Yaskawa INFORM job: X2_48(150,-90).JBI

/JOB
//NAME X2_48(150,-90)
//POS
///NPOS 103,103,103,5,0,0
///TOOL 0
///POSTYPE PULSE
///PULSE
C00000=-2000,-112988,-119327,0,83158,0
C00001=142756,-112988,-119327,18089,83158,-34222
C00002=145489,-137180,-128771,21394,87700,-32111
C00003=164591,-94889,-79086,18920,74682,-27376
C00004=167906,-89992,-74155,18360,73432,-26351
C00005=169175,-88015,-72150,18139,72941,-25959
C00006=169090,-86796,-69106,18271,71772,-26171
C00007=169175,-88015,-72150,18139,72941,-25959
C00008=170099,-88727,-72164,17993,72396,-25701
C00009=172764,-85592,-70856,17391,72586,-24688
C00010=170099,-88727,-72164,17993,72396,-25701
C00011=185420,-95958,-68594,-7326,50076,-11474
C00012=182716,-92695,-67464,-5857,50831,-12695
C00013=185420,-95958,-68594,-7326,50076,-11474
C00014=184506,-107402,-76413,-6968,48935,-11790
C00015=159220,-109944,-102922,24512,66979,-45642
C00016=167824,-173568,-124205,26542,46564,-47026
C00017=170252,-85554,-47492,36176,17718,-77515
C00018=172784,-79149,-41877,32040,16598,-75352
C00019=173728,-77240,-40780,29717,16528,-74186
C00020=176622,-74360,-39545,22774,16291,-70707
C00021=173728,-77240,-40780,29717,16528,-74186
C00022=175036,-75947,-40158,26684,16349,-72661
C00023=174520,-73484,-36544,29303,15665,-73921
C00024=175036,-76518,-41235,26130,16681,-72405
C00025=171703,-84374,-47061,33102,17430,-75946
C00026=118222,-104921,-85597,-2302,76232,3756
C00027=70971,-85923,-48405,-35291,17571,76879
C00028=68458,-79485,-42811,-31017,16504,74660
C00029=67521,-76918,-40527,-29335,16103,73795
C00030=65747,-75173,-39789,-24982,15938,71620
C00031=67521,-76918,-40527,-29335,16103,73795
C00032=66355,-75782,-40029,-26507,15971,72380
C00033=66862,-73889,-37487,-28530,15606,73362
C00034=66355,-75782,-40029,-26507,15971,72380
C00035=67257,-78357,-42329,-28198,16341,73244
C00036=69676,-84817,-47961,-32519,17317,75468
C00037=66595,-165951,-119904,-20395,34837,49941
C00038=38828,-178555,-122254,18105,43219,2401
C00039=76877,-95412,-79683,-19208,74450,27234
C00040=73543,-90451,-74757,-18629,73220,26200
C00041=72268,-88450,-72755,-18400,72736,25804
C00042=72333,-87219,-69709,-18531,71571,26012
C00043=72268,-88450,-72755,-18400,72736,25804
C00044=71656,-87743,-71624,-18310,72282,25648
C00045=69017,-84617,-70326,-17702,72469,24642
C00046=71656,-87743,-71624,-18310,72282,25648
C00047=55558,-95793,-69122,7502,50260,11083
C00048=58281,-92556,-67996,6016,50996,12311
C00049=55558,-95793,-69122,7502,50260,11083
C00050=56403,-107290,-76939,7182,49095,11365
C00051=66823,-91712,-74133,-7065,60566,19717
C00052=66824,-90415,-70771,-7163,59174,19807
C00053=66853,-89833,-69254,-7221,58546,19861
C00054=63349,-96192,-73367,-19942,70973,24588
C00055=64655,-93749,-71616,-22869,75239,26164
C00056=62828,-96481,-72572,-22743,73980,25724
C00057=62157,-97058,-72609,-22694,73543,25556
C00058=66824,-90716,-71530,-22972,77234,26586
C00059=66823,-92043,-75030,-22863,78594,26321
C00060=119458,-64652,-78063,-7993,91912,2412
C00061=162081,-130804,-92299,12648,53591,-25594
C00062=176554,-94726,-71925,6352,57827,-19319
C00063=177319,-91851,-69580,6047,57801,-19017
C00064=164142,-69963,-61844,21170,80838,-28219
C00065=180939,-101074,-74209,19420,68796,-24064
C00066=178968,-96927,-72415,22445,73972,-25771
C00067=182294,-101580,-74047,22207,71788,-24939
C00068=185323,-105159,-75046,21972,69843,-24161
C00069=177337,-98931,-74291,22610,74536,-26275
C00070=148639,-128504,-104999,23996,86118,-34643
C00071=125763,-70435,-126192,-3026,94587,28672
C00072=71267,-74397,-112769,20427,89435,13482
C00073=68499,-138788,-124688,-10863,39680,60380
C00074=66279,-93192,-102590,-7723,49796,58218
C00075=64635,-80465,-95998,-4093,52558,56280
C00076=64736,-80204,-95947,-4166,52664,56317
C00077=66642,-84423,-98093,-16099,53671,64179
C00078=66744,-83933,-97854,-14906,51366,64983
C00079=66851,-84061,-98003,-13231,47738,66189
C00080=66924,-84097,-98180,-11670,44122,67370
C00081=67067,-84256,-98352,-9466,37843,69430
C00082=62617,-94836,-103731,-1077,27723,69260
C00083=60476,-99306,-104126,2746,25300,67760
C00084=58396,-103594,-105732,6580,24205,66047
C00085=71788,-113583,-131480,-12468,38511,72889
C00086=126548,-133354,-124162,-3479,55623,10129
C00087=185990,-110059,-108050,2198,41333,-59059
C00088=176703,-90185,-100504,9996,47566,-62974
C00089=174384,-84529,-98133,11690,49287,-63786
C00090=174879,-80146,-95973,11134,50130,-63480
C00091=175328,-83211,-97701,10847,49566,-63351
C00092=176891,-87663,-99301,14966,53867,-62708
C00093=175291,-82874,-97472,15103,53157,-64529
C00094=175284,-82851,-97494,13305,49526,-65702
C00095=175317,-82765,-97451,12150,47080,-66463
C00096=175369,-82638,-97277,9095,39505,-68806
C00097=177670,-88810,-99810,5702,34313,-68809
C00098=179386,-92866,-101274,2581,30714,-68509
C00099=180987,-99716,-104277,-2046,25458,-68211
C00100=183030,-103926,-105848,-5755,24360,-66553
C00101=165604,-146579,-119354,35431,57728,-66075
C00102=-2000,-112988,-119327,0,83158,0
BC00000=91885,523905,1075139
BC00001=176516,513386,1075139
BC00002=176516,372432,1075139
BC00003=176516,372432,1075139
BC00004=176516,372432,1075139
BC00005=176516,372432,1075139
BC00006=176516,372432,1075139
BC00007=176516,372432,1075139
BC00008=176516,372432,1075139
BC00009=176516,372432,1075139
BC00010=176516,372432,1075139
BC00011=176516,372432,1075139
BC00012=176516,372432,1075139
BC00013=176516,372432,1075139
BC00014=176516,372432,1075139
BC00015=185933,410402,1075139
BC00016=185933,426050,1075139
BC00017=201871,474658,1075139
BC00018=201871,474658,1075139
BC00019=201871,474658,1075139
BC00020=201871,474658,1075139
BC00021=201871,474658,1075139
BC00022=201871,474658,1075139
BC00023=201871,474658,1075139
BC00024=201871,474658,1075139
BC00025=201871,474658,1075139
BC00026=220143,474168,1075139
BC00027=236265,473735,1075139
BC00028=236265,473735,1075139
BC00029=236265,473735,1075139
BC00030=236265,473735,1075139
BC00031=236265,473735,1075139
BC00032=236265,473735,1075139
BC00033=236265,473735,1075139
BC00034=236265,473735,1075139
BC00035=236265,473735,1075139
BC00036=220985,493295,1073179
BC00037=243232,450879,1070770
BC00038=260102,370644,1075139
BC00039=260102,370644,1075139
BC00040=260102,370644,1075139
BC00041=260102,370644,1075139
BC00042=260102,370644,1075139
BC00043=260102,370644,1075139
BC00044=260102,370644,1075139
BC00045=260102,370644,1075139
BC00046=260102,370644,1075139
BC00047=260102,370644,1075139
BC00048=260102,370644,1075139
BC00049=260102,370644,1075139
BC00050=260102,370644,1075139
BC00051=256587,368878,1075139
BC00052=262038,366660,1075139
BC00053=264218,365773,1075139
BC00054=261883,337583,1075139
BC00055=262912,371200,1075139
BC00056=262912,371200,1075139
BC00057=262912,371200,1075139
BC00058=260684,370761,1075139
BC00059=255114,369664,1075139
BC00060=215679,440004,1075139
BC00061=173780,363609,1075139
BC00062=173780,363609,1075139
BC00063=173780,363609,1075139
BC00064=173780,363609,1075139
BC00065=173780,363609,1075139
BC00066=173780,363609,1075139
BC00067=173780,363609,1075139
BC00068=173780,363609,1075139
BC00069=173780,363609,1075139
BC00070=173780,363609,1075139
BC00071=206768,500109,907660
BC00072=206768,522353,907660
BC00073=237122,456071,765063
BC00074=234854,454602,775976
BC00075=235225,454500,774776
BC00076=235225,454500,774776
BC00077=230684,451767,767257
BC00078=230752,464387,749473
BC00079=230835,478504,722885
BC00080=230942,495701,685005
BC00081=231085,514573,626364
BC00082=231233,523596,542063
BC00083=228995,523889,543694
BC00084=223383,523889,557697
BC00085=223369,523889,578107
BC00086=226901,519330,831694
BC00087=230821,475079,776375
BC00088=212990,455632,776375
BC00089=207393,454117,758000
BC00090=206067,453758,753645
BC00091=205154,453511,750649
BC00092=206622,445635,770734
BC00093=207343,466946,745914
BC00094=207413,478057,723264
BC00095=207497,491870,694918
BC00096=207664,515607,624377
BC00097=207731,518542,592641
BC00098=207778,520613,570250
BC00099=210096,523889,540489
BC00100=215706,523889,554630
BC00101=215706,523889,928949
BC00102=91885,523905,1075139
EC00000=-1330261,372643
EC00001=-1330261,372643
EC00002=-1330261,372643
EC00003=-1330261,372643
EC00004=-1330261,372643
EC00005=-1330261,372643
EC00006=-1330261,372643
EC00007=-1330261,372643
EC00008=-1330261,372643
EC00009=-1330261,372643
EC00010=-1330261,372643
EC00011=-1330261,372643
EC00012=-1330261,372643
EC00013=-1330261,372643
EC00014=-1330261,372643
EC00015=-1330261,372643
EC00016=-1330261,372643
EC00017=-1330261,372643
EC00018=-1330261,372643
EC00019=-1330261,372643
EC00020=-1330261,372643
EC00021=-1330261,372643
EC00022=-1330261,372643
EC00023=-1330261,372643
EC00024=-1330261,372643
EC00025=-1330261,372643
EC00026=-1330261,372643
EC00027=-1330261,372643
EC00028=-1330261,372643
EC00029=-1330261,372643
EC00030=-1330261,372643
EC00031=-1330261,372643
EC00032=-1330261,372643
EC00033=-1330261,372643
EC00034=-1330261,372643
EC00035=-1330261,372643
EC00036=-1330261,372643
EC00037=-1330261,372643
EC00038=-1330261,372643
EC00039=-1330261,372643
EC00040=-1330261,372643
EC00041=-1330261,372643
EC00042=-1330261,372643
EC00043=-1330261,372643
EC00044=-1330261,372643
EC00045=-1330261,372643
EC00046=-1330261,372643
EC00047=-1330261,372643
EC00048=-1330261,372643
EC00049=-1330261,372643
EC00050=-1330261,372643
EC00051=-1330261,372643
EC00052=-1330261,372643
EC00053=-1330261,372643
EC00054=-1330261,372643
EC00055=-1330261,372643
EC00056=-1330261,372643
EC00057=-1330261,372643
EC00058=-1330261,372643
EC00059=-1330261,372643
EC00060=-1330261,372643
EC00061=-1330261,372643
EC00062=-1330261,372643
EC00063=-1330261,372643
EC00064=-1330261,372643
EC00065=-1330261,372643
EC00066=-1330261,372643
EC00067=-1330261,372643
EC00068=-1330261,372643
EC00069=-1330261,372643
EC00070=-1330261,372643
EC00071=-1330261,372643
EC00072=-1330261,372643
EC00073=-1330261,372643
EC00074=-1330261,372643
EC00075=-1330261,372643
EC00076=-1330261,372643
EC00077=-1330261,372643
EC00078=-1330261,372643
EC00079=-1330261,372643
EC00080=-1330261,372643
EC00081=-1330261,372643
EC00082=-1330261,372643
EC00083=-1330261,372643
EC00084=-1330261,372643
EC00085=-1330261,372643
EC00086=-1330261,372643
EC00087=-1330261,372643
EC00088=-1330261,372643
EC00089=-1330261,372643
EC00090=-1330261,372642
EC00091=-1330261,372643
EC00092=-1330261,372643
EC00093=-1330261,372643
EC00094=-1330261,372643
EC00095=-1330261,372643
EC00096=-1330261,372643
EC00097=-1330261,372643
EC00098=-1330261,372643
EC00099=-1330261,372643
EC00100=-1330261,372643
EC00101=-1330261,372643
EC00102=-1330261,372643
///POSTYPE BASE
///RECTAN
///RCONF 0,0,0,0,1,0,0,0,0,0,0,0,0,0,0,0,0,0,0,0,0,0,0,0
P00006=2.006,1.622,-0.565,0.0000,0.0000,0.0000
P00021=0.073,2.058,-0.109,0.0000,0.0000,0.0000
P00022=2.006,1.622,-0.565,0.0000,0.0000,0.0000
///RCONF 0,0,0,0,0,0,0,0,0,0,0,0,0,0,0,0,0,0,0,0,0,0,0,0
P00031=-0.170,0.039,-0.647,0.0000,0.0000,0.0000
P00032=-0.423,0.157,3.222,0.0000,0.0000,0.0000
//INST
///DATE 2024/12/19 12:01
///ATTR SC,RW
///GROUP1 RB1,BS1
///GROUP2 ST1
NOP
'X2_48(150,-90)
MOVJ C00000 BC00000 VJ=100.00  +MOVJ EC00000 VJ=100.00
MOVJ C00001 BC00001 VJ=100.00  +MOVJ EC00001 VJ=100.00
MOVJ C00002 BC00002 VJ=100.00  +MOVJ EC00002 VJ=100.00
'Path S3695
SFTOF3D
MOVJ C00003 BC00003 VJ=100.00  +MOVJ EC00003 VJ=100.00
MOVL C00004 BC00004 V=800.0  +MOVJ EC00004 VJ=100.00
SMOVL C00005 BC00005 V=166.7  +MOVJ EC00005
SREFP 3 C00006 BC00006  +REFP EC00006
CALL JOB:SEARCH-R1-S13D
SET P032 P006
SFTON3D P032
SMOVL C00007 BC00007 V=166.7  +MOVJ EC00007
SMOVL C00008 BC00008 V=166.7  +MOVJ EC00008
SREFP 3 C00009 BC00009  +REFP EC00009
CALL JOB:SEARCH-R1-S13D
SET P032 P006
SFTON3D P032
SMOVL C00010 BC00010 V=166.7  +MOVJ EC00010
SMOVL C00011 BC00011 V=166.7  +MOVJ EC00011
SREFP 3 C00012 BC00012  +REFP EC00012
CALL JOB:SEARCH-R1-S13D
SET P032 P006
SFTON3D P032
SMOVL C00013 BC00013 V=166.7  +MOVJ EC00013
MOVL C00014 BC00014 V=1000.0  +MOVJ EC00014 VJ=100.00
'EndPath S3695
MOVJ C00015 BC00015 VJ=100.00  +MOVJ EC00015 VJ=100.00
MOVJ C00016 BC00016 VJ=100.00  +MOVJ EC00016 VJ=100.00
'Path S3694
SFTOF3D
MOVJ C00017 BC00017 VJ=100.00  +MOVJ EC00017 VJ=100.00
MOVL C00018 BC00018 V=800.0  +MOVJ EC00018 VJ=100.00
SMOVL C00019 BC00019 V=166.7  +MOVJ EC00019
SREFP 3 C00020 BC00020  +REFP EC00020
CALL JOB:SEARCH-R1-S13D
SET P022 P006
SFTON3D P022
SMOVL C00021 BC00021 V=166.7  +MOVJ EC00021
SMOVL C00022 BC00022 V=166.7  +MOVJ EC00022
SREFP 3 C00023 BC00023  +REFP EC00023
CALL JOB:SEARCH-R1-S13D
SET P022 P006
SFTON3D P022
SMOVL C00024 BC00024 V=166.7  +MOVJ EC00024
MOVL C00025 BC00025 V=1000.0  +MOVJ EC00025 VJ=100.00
'EndPath S3694
MOVJ C00026 BC00026 VJ=100.00  +MOVJ EC00026 VJ=100.00
'Path S3696
SFTOF3D
MOVJ C00027 BC00027 VJ=100.00  +MOVJ EC00027 VJ=100.00
MOVL C00028 BC00028 V=800.0  +MOVJ EC00028 VJ=100.00
SMOVL C00029 BC00029 V=166.7  +MOVJ EC00029
SREFP 3 C00030 BC00030  +REFP EC00030
CALL JOB:SEARCH-R1-S13D
SET P021 P006
SFTON3D P021
SMOVL C00031 BC00031 V=166.7  +MOVJ EC00031
SMOVL C00032 BC00032 V=166.7  +MOVJ EC00032
SREFP 3 C00033 BC00033  +REFP EC00033
CALL JOB:SEARCH-R1-S13D
SET P021 P006
SFTON3D P021
SMOVL C00034 BC00034 V=166.7  +MOVJ EC00034
MOVL C00035 BC00035 V=800.0  +MOVJ EC00035 VJ=100.00
MOVL C00036 BC00036 V=1000.0  +MOVJ EC00036 VJ=100.00
'EndPath S3696
MOVJ C00037 BC00037 VJ=100.00  +MOVJ EC00037 VJ=100.00
MOVJ C00038 BC00038 VJ=100.00  +MOVJ EC00038 VJ=100.00
'Path S3697
SFTOF3D
MOVJ C00039 BC00039 VJ=100.00  +MOVJ EC00039 VJ=100.00
MOVL C00040 BC00040 V=800.0  +MOVJ EC00040 VJ=100.00
SMOVL C00041 BC00041 V=166.7  +MOVJ EC00041
SREFP 3 C00042 BC00042  +REFP EC00042
CALL JOB:SEARCH-R1-S13D
SET P031 P006
SFTON3D P031
SMOVL C00043 BC00043 V=166.7  +MOVJ EC00043
SMOVL C00044 BC00044 V=166.7  +MOVJ EC00044
SREFP 3 C00045 BC00045  +REFP EC00045
CALL JOB:SEARCH-R1-S13D
SET P031 P006
SFTON3D P031
SMOVL C00046 BC00046 V=166.7  +MOVJ EC00046
SMOVL C00047 BC00047 V=166.7  +MOVJ EC00047
SREFP 3 C00048 BC00048  +REFP EC00048
CALL JOB:SEARCH-R1-S13D
SET P031 P006
SFTON3D P031
SMOVL C00049 BC00049 V=166.7  +MOVJ EC00049
MOVL C00050 BC00050 V=1000.0  +MOVJ EC00050 VJ=100.00
'EndPath S3697
'Path W3698
SFTOF3D
SFTON3D P031
MOVJ C00051 BC00051 VJ=100.00  +MOVJ EC00051 VJ=100.00
SMOVL C00052 BC00052 V=800.0  +MOVJ EC00052
SMOVL C00053 BC00053 V=166.7 PL=0  +MOVJ EC00053
MACRO1 MJ#(0) ARGF22
ARCON
SMOVL C00054 BC00054 V=10.0  +MOVJ EC00054
SMOVL C00055 BC00055 V=10.0  +MOVJ EC00055
SMOVL C00056 BC00056 V=10.0  +MOVJ EC00056
SMOVL C00057 BC00057 V=10.0  +MOVJ EC00057
ARCOF
SMOVL C00058 BC00058 V=800.0  +MOVJ EC00058
SMOVL C00059 BC00059 V=1000.0  +MOVJ EC00059
SFTOF3D
'EndPath W3698
MOVJ C00060 BC00060 VJ=100.00  +MOVJ EC00060 VJ=100.00
'Path W3699
SFTOF3D
SFTON3D P032
MOVJ C00061 BC00061 VJ=100.00  +MOVJ EC00061 VJ=100.00
SMOVL C00062 BC00062 V=800.0  +MOVJ EC00062
SMOVL C00063 BC00063 V=166.7 PL=0  +MOVJ EC00063
ARCON
SMOVL C00064 BC00064 V=10.0  +MOVJ EC00064
SMOVL C00065 BC00065 V=10.0  +MOVJ EC00065
SMOVL C00066 BC00066 V=10.0  +MOVJ EC00066
SMOVL C00067 BC00067 V=10.0  +MOVJ EC00067
SMOVL C00068 BC00068 V=10.0  +MOVJ EC00068
ARCOF
SMOVL C00069 BC00069 V=800.0  +MOVJ EC00069
MOVJ C00070 BC00070 VJ=100.00  +MOVJ EC00070 VJ=100.00
SFTOF3D
'EndPath W3699
MOVJ C00071 BC00071 VJ=100.00  +MOVJ EC00071 VJ=100.00
MOVJ C00072 BC00072 VJ=100.00  +MOVJ EC00072 VJ=100.00
MOVJ C00073 BC00073 VJ=100.00  +MOVJ EC00073 VJ=100.00
'Path W3700
SFTOF3D
SFTON3D P021
SMOVL C00074 BC00074 V=800.0  +MOVJ EC00074
SMOVL C00075 BC00075 V=333.3  +MOVJ EC00075
ARCON
SMOVC C00076 BC00076 V=10.0  +MOVJ EC00076
SMOVC C00077 BC00077 V=10.0  +MOVJ EC00077
SMOVC C00078 BC00078 V=10.0  +MOVJ EC00078
SMOVC C00079 BC00079 V=10.0  +MOVJ EC00079
SMOVC C00080 BC00080 V=10.0  +MOVJ EC00080
SMOVC C00081 BC00081 V=10.0  +MOVJ EC00081
SMOVC C00082 BC00082 V=10.0  +MOVJ EC00082
ARCOF
SMOVL C00083 BC00083 V=800.0  +MOVJ EC00083
SMOVL C00084 BC00084 V=1000.0  +MOVJ EC00084
SFTOF3D
'EndPath W3700
MOVJ C00085 BC00085 VJ=100.00  +MOVJ EC00085 VJ=100.00
MOVJ C00086 BC00086 VJ=100.00  +MOVJ EC00086 VJ=100.00
MOVJ C00087 BC00087 VJ=100.00  +MOVJ EC00087 VJ=100.00
'Path W4285
SFTOF3D
SFTON3D P022
MOVJ C00088 BC00088 VJ=100.00  +MOVJ EC00088 VJ=100.00
SMOVL C00089 BC00089 V=800.0  +MOVJ EC00089
SMOVC C00090 BC00090 V=150.0 PL=0  +MOVJ EC00090
ARCON
SMOVC C00091 BC00091 V=10.0  +MOVJ EC00091
SMOVC C00092 BC00092 V=10.0  +MOVJ EC00092
SMOVC C00093 BC00093 V=10.0  +MOVJ EC00093
SMOVC C00094 BC00094 V=10.0  +MOVJ EC00094
SMOVC C00095 BC00095 V=10.0  +MOVJ EC00095
SMOVC C00096 BC00096 V=10.0  +MOVJ EC00096
SMOVC C00097 BC00097 V=10.0  +MOVJ EC00097
SMOVL C00098 BC00098 V=10.0  +MOVJ EC00098
ARCOF
SMOVL C00099 BC00099 V=800.0  +MOVJ EC00099
SMOVL C00100 BC00100 V=1000.0  +MOVJ EC00100
SFTOF3D
'EndPath W4285
MOVJ C00101 BC00101 VJ=100.00  +MOVJ EC00101 VJ=100.00
MOVJ C00102 BC00102 VJ=100.00  +MOVJ EC00102 VJ=100.00
END
